# B&R Automation Studio project ai_powered_plc_development
Automation Studio 6.3.1.32; technology packages: mappConnect 6.1.0, mappView 6.1.1, OpcUaCs 6.0.0

## Configuration Main

CPU X20CP1686X, AutomationRuntime 6.3.3, Build 11.3.0, Vc 6.0.0

### Task classes (Cpu.sw)
```
Cyclic#1:
  method <- Method.method.prg
Cyclic#4:
  mco <- mco.prg
  Main <- Source.Main.prg
  Conveyor <- Source.Modules.Conveyor.Conveyor.prg
  Heater <- Source.Modules.Heater.Heater.prg
  Robot <- Source.Modules.Robot.Robot.prg
  AlarmHandl <- Source.Services.AlarmHandler.AlarmHandler.prg
Libraries: CoTrace, runtime, AsZip, FileIO, AsOpcUac, AsOpcUas
```

### Hardware
```
X20CP1686X : X20CP1686X v1.8.2.0
  Connector IF2:
    ActivateDevice = 1
  ConfigurationID = ai_powered_plc_development_mappConnectDemo
  AutomaticTransferOfUserfiles = on
  FileDevice1
  FileDeviceName1 = USER
  FileDevicePath1 = USER_PATH
  FileDevice2
  FileDeviceName2 = USER_web
  FileDevicePath2 = USER_PATH/web
  ActivateWebServer = 1
  WebServerProtocol = 1
```

### Config.mappconnect - X20CP1686X/mappConnect/Config.mappconnect
```
Element mapp Connect Configuration (Type=mappconnect)
  WebServerProtocol = 1
    WebServerPort = 8080
    Interface = All
    WebServerPortSsl = 8443
  WebServerEndpointConfiguration:
    Endpoint[1]  // Allow .html files for all users
      Endpoint = *.html
      Roles
    Endpoint[2]  // Allow stylesheet files for all users
      Endpoint = /css/*.css
      Roles
    Endpoint[3]  // Allow javascript files for all users
      Endpoint = /js/*.js
      Roles
    Endpoint[4]  // Allow all API endpoints for all users
      Endpoint = /api/1.0/*
      Roles
    Endpoint[5]  // Allow favicon and icon files
      Endpoint = *.ico
      Roles
    Endpoint[6]  // Allow common image types
      Endpoint = *.png
      Roles
    Endpoint[7]  // Allow common image types
      Endpoint = *.jpg
      Roles
    Endpoint[8]  // Allow common image types
      Endpoint = *.svg
      Roles
    Endpoint[9]  // Allow fonts
      Endpoint = *.woff2
      Roles
    Endpoint[10]  // Allow fonts
      Endpoint = *.woff
      Roles
    Endpoint[11]  // Allow fonts
      Endpoint = *.ttf
      Roles
    Endpoint[12]  // Allow source maps (dev)
      Endpoint = *.map
      Roles
    Endpoint[13]  // Allow typical asset folders
      Endpoint = /assets/*
      Roles
    Endpoint[14]  // Allow typical image folder
      Endpoint = /img/*
      Roles
    Endpoint[15]  // Allow additional static folder
      Endpoint = /static/*
      Roles
  OpcUaServerWhitelist:
    OpcUaServer[1]:
      Url = opc.tcp://127.0.0.1:4840
```

### AlarmCore.mpalarmxcore - X20CP1686X/mappServices/AlarmCore.mpalarmxcore
```
Element gAlarmXCore (Type=mpalarmxcore)
  mapp.Gen:
    Enable = TRUE
    EnableCockpit = TRUE
    TaskClass = 4
    Parent
  mapp.AlarmX.List:
    [0]:
      List = gAlarmXList
      Offset = 0
  mapp.AlarmX.Create = Disabled
  mapp.AlarmX.Core.Retain:
    Memory = 0
  mapp.AlarmX.Core.Categories:
    [0]:
      List = gAlarmXCategory
```

### AlarmHist.mpalarmxhistory - X20CP1686X/mappServices/AlarmHist.mpalarmxhistory
```
Element gAlarmXHistory (Type=mpalarmxhistory)
  mapp.Gen:
    Enable = TRUE
    EnableCockpit = TRUE
    Audit = TRUE
    Parent
  mapp.AlarmX.History:
    Export:
      TimeStampPattern = %Y-%m-%d %H:%M:%S:%L
      AutoExtension = TRUE
      ColumnSeparator = ,
    Memory = 0
      Size = 200
      BufferSize = 10
      Interval = 60
    Scope = 0
```

### AlarmList.mpalarmxlist - X20CP1686X/mappServices/AlarmList.mpalarmxlist
```
Element gAlarmXList (Type=mpalarmxlist)
  mapp.AlarmX.Snippets:
    AutoDetect = 1
      Language
```

## Logical view

Binary libraries used (declarations not repeated): operator, runtime, AsIecCon, astime, CoTrace, AsZip, FileIO, AsOpcUac, AsOpcUas


### Program Logical/mco (ANSIC)

#### Variables.var
```iecst
VAR
	myVar : LREAL := 12.3;
	myVar2 : REAL := 11;
END_VAR
```

#### compile_flags.txt
```
# This file is auto-generated by ASX. Do not edit manually, as changes may be overwritten.
# If you need to manually edit this file and prevent automatic updates, add "# MANUAL EDIT" to the first line.
-I
c:\projects\Private\ai_powered_plc_development\Logical\mco
-I
c:\projects\Private\ai_powered_plc_development\Temp\Includes\mco
-I
C:\Program Files (x86)\BRAutomation\AS6\AS\gnuinst\V11.3.0\6.0\i686-elf\include\c++\11.3.0
-I
C:\Program Files (x86)\BRAutomation\AS6\AS\gnuinst\V11.3.0\6.0\i686-elf\include\c++\11.3.0\i686-elf
-I
C:\Program Files (x86)\BRAutomation\AS6\AS\gnuinst\V11.3.0\6.0\i686-elf\include\c++\11.3.0\backward
-I
C:\Program Files (x86)\BRAutomation\AS6\AS\gnuinst\V11.3.0\6.0\lib\gcc\i686-elf\11.3.0\include
-I
C:\Program Files (x86)\BRAutomation\AS6\AS\gnuinst\V11.3.0\6.0\lib\gcc\i686-elf\11.3.0\include-fixed
-I
C:\Program Files (x86)\BRAutomation\AS6\AS\gnuinst\V11.3.0\6.0\i686-elf\include
-I
c:\projects\Private\ai_powered_plc_development\Temp\Includes
-trigraphs
-fno-asm
-D
_DEFAULT_INCLUDES
-D
_SG4
--target=i686-elf
-fPIC
-Wall
```

#### Cyclic.c
```c
#include <bur/plctypes.h>

#ifdef _DEFAULT_INCLUDES
	#include <AsDefault.h>
#endif

void _CYCLIC ProgramCyclic(void)
{

}
```

### Program Logical/Method/method (ANSIC)

#### Cyclic.c - Cyclic code
```c
#include <bur/plctypes.h>

#ifdef _DEFAULT_INCLUDES
	#include <AsDefault.h>
#endif

#include <string.h>

void _CYCLIC ProgramCyclic(void)
{
	switch(state)
	{
		case WaitForCall:
			UaSrv_MethodOperate_0.Action = UaMoa_CheckIsCalled;
			UaSrv_MethodOperate(&UaSrv_MethodOperate_0);
			UaSrv_MethodOperate_0.Execute = !UaSrv_MethodOperate_0.Busy;
			if (UaSrv_MethodOperate_0.Done && UaSrv_MethodOperate_0.IsCalled)
			{
				state = ExecuteMethod;
			}
			if (UaSrv_MethodOperate_0.Error)
			{
				state = Error;
			}
			break;

		case ExecuteMethod:
			methodCalled = 1;
			output1 = input1 + input2;
			state = FinishMethod;
			UaSrv_MethodOperate_0.Execute = 1;
			break;

		case FinishMethod:
			UaSrv_MethodOperate_0.Action = UaMoa_Finished;
			UaSrv_MethodOperate(&UaSrv_MethodOperate_0);
			UaSrv_MethodOperate_0.Execute = !UaSrv_MethodOperate_0.Busy;
			if (UaSrv_MethodOperate_0.Done)
			{
				state = WaitForCall;
			}
			if (UaSrv_MethodOperate_0.Error)
			{
				state = Error;
			}
			break;

		case Error:
			break;

		default:
			state = Error;
	}
}
```

#### Types.typ - Local data types
```iecst
TYPE
	State :
		(
		WaitForCall,
		ExecuteMethod,
		FinishMethod,
		Error
		);
END_TYPE
```

#### Variables.var - Local variables
```iecst
VAR
	output1 : DINT;
	input1 : DINT;
	UaSrv_MethodOperate_0 : UaSrv_MethodOperate;
	state : State := WaitForCall;
END_VAR
VAR CONSTANT
	cMethodName : STRING[32] := 'add';
END_VAR
VAR
	methodCalled : BOOL := FALSE;
	input2 : DINT;
END_VAR
```

- Methods.uam (not shown)

#### Init.c - Initialization code
```c
#include <bur/plctypes.h>

#ifdef _DEFAULT_INCLUDES
	#include <AsDefault.h>
#endif

#include <string.h>

void _INIT ProgramInit(void)
{
	strcpy(UaSrv_MethodOperate_0.MethodName, cMethodName);
}
```

### MainIface.typ
```iecst
TYPE
	MainCmdIfaceType : STRUCT
		Start : BOOL;
		Stop  : BOOL;
	END_STRUCT;

	MainParIfaceType : STRUCT
		Reserved : BOOL;
	END_STRUCT;

	MainStatusIfaceType : STRUCT
		State       : STRING[32];
		Substate    : STRING[32];
		LineRunning : BOOL;
		AnyFault    : BOOL;
	END_STRUCT;

	MainIfaceType : STRUCT
		Cmd    : MainCmdIfaceType;
		Par    : MainParIfaceType;
		Status : MainStatusIfaceType;
	END_STRUCT;
END_TYPE
```

### MainIface.var
```iecst
VAR
	gMain : MainIfaceType;
END_VAR

VAR CONSTANT

END_VAR
```

### Types.typ
```iecst
TYPE
	(* HMI data transfer objects for Main aggregate *)

	ConveyorHmiData : STRUCT
		Running    : BOOL;
		Fault      : BOOL;
		Speed      : REAL;      (* m/s *)
		Load       : REAL;      (* % *)
		PartsCount : UDINT;
		Mode       : STRING[16];
	END_STRUCT;

	HeaterHmiData : STRUCT
		Heating      : BOOL;
		Fault        : BOOL;
		Temperature  : REAL;     (* °C *)
		PowerPercent : REAL;     (* % *)
		Setpoint     : REAL;     (* °C *)
	END_STRUCT;

	RobotHmiData : STRUCT
		Auto  : BOOL;
		Fault : BOOL;
		X     : REAL;
		Y     : REAL;
		Z     : REAL;
		State : STRING[32];
	END_STRUCT;

	MachineCommandsType : STRUCT
		Start : BOOL;
		Stop  : BOOL;
	END_STRUCT;

	MachineHmiData : STRUCT
		State       : STRING[32];
		Substate    : STRING[64];
		LineRunning : BOOL;
		AnyFault    : BOOL;
		Conveyor    : ConveyorHmiData;
		Heater      : HeaterHmiData;
		Robot       : RobotHmiData;
		Commands    : MachineCommandsType;
	END_STRUCT;

END_TYPE
```

### Variables.var
```iecst
VAR
    MachineHmi : MachineHmiData; (* Exposed HMI aggregate *)
    runRequest : BOOL; (* internal latched run flag *)
END_VAR

VAR CONSTANT

END_VAR
```

### MainIface.typ - not listed in the package file held
```iecst
TYPE
    MainCmdIfaceType : STRUCT
        Start : BOOL;
        Stop  : BOOL;
    END_STRUCT;

    MainParIfaceType : STRUCT
        Reserved : BOOL;
    END_STRUCT;

    MainStatusIfaceType : STRUCT
        State     : STRING[32];
        Substate  : STRING[32];
        LineRunning : BOOL;
        AnyFault    : BOOL;
    END_STRUCT;

    MainIfaceType : STRUCT
        Cmd    : MainCmdIfaceType;
        Par    : MainParIfaceType;
        Status : MainStatusIfaceType;
    END_STRUCT;
END_TYPE
```

### MainIface.var - not listed in the package file held
```iecst
VAR
    gMain : MainIfaceType;
END_VAR

VAR CONSTANT
END_VAR
```

### Main.st - not listed in the package file held
```iecst
PROGRAM _INIT
	(* Insert code here *)
	(* Initialize defaults *)
	MachineHmi.LineRunning := FALSE;
	MachineHmi.State := 'Idle';
	MachineHmi.Substate := '';
	runRequest := FALSE;
	(* Initialize main interface status *)
	gMain.Status.State := 'Idle';
	gMain.Status.Substate := '';
	gMain.Status.LineRunning := FALSE;
	gMain.Status.AnyFault := FALSE;
END_PROGRAM

PROGRAM _CYCLIC
	(* Pull conveyor status from its program interface *)
	MachineHmi.Conveyor.Running := gConveyor.Status.Running;
	MachineHmi.Conveyor.Fault := gConveyor.Status.Fault;
	MachineHmi.Conveyor.Speed := gConveyor.Status.Speed_mps;
	MachineHmi.Conveyor.Load := gConveyor.Status.Load_pct;
	MachineHmi.Conveyor.PartsCount := gConveyor.Status.PartsCount;
	MachineHmi.Conveyor.Mode := gConveyor.Status.Mode;

	(* Heater status from module interface *)
	MachineHmi.Heater.Heating := gHeater.Status.Heating;
	MachineHmi.Heater.Fault := gHeater.Status.Fault;
	MachineHmi.Heater.Temperature := gHeater.Status.TemperatureC;
	MachineHmi.Heater.PowerPercent := gHeater.Status.Power_pct;
	IF gHeater.Par.Setpoint_C <> 0.0 THEN MachineHmi.Heater.Setpoint := gHeater.Par.Setpoint_C; END_IF;

	(* Robot status from module interface *)
	MachineHmi.Robot.Auto := gRobot.Status.Auto;
	MachineHmi.Robot.Fault := gRobot.Status.Fault;
	MachineHmi.Robot.X := gRobot.Status.X;
	MachineHmi.Robot.Y := gRobot.Status.Y;
	MachineHmi.Robot.Z := gRobot.Status.Z;
	MachineHmi.Robot.State := gRobot.Status.State;

	(* Aggregate HMI level flags *)
	MachineHmi.AnyFault := MachineHmi.Conveyor.Fault OR MachineHmi.Heater.Fault OR MachineHmi.Robot.Fault;
	MachineHmi.LineRunning := runRequest AND NOT MachineHmi.AnyFault;

	(* Interfaces already mapped above *)

	(* Determine State/Substate *)
	IF MachineHmi.AnyFault THEN
		MachineHmi.State := 'Fault';
		MachineHmi.Substate := 'Check modules';
	ELSIF runRequest THEN
		MachineHmi.State := 'Auto';
		IF NOT gConveyor.Status.Running THEN
			MachineHmi.Substate := 'Starting conveyor';
		ELSIF NOT gRobot.Status.Auto THEN
			MachineHmi.Substate := 'Starting robot';
		ELSE
			MachineHmi.Substate := 'Production';
		END_IF;
	ELSE
		MachineHmi.State := 'Idle';
		MachineHmi.Substate := 'Waiting for start';
	END_IF;

	(* Process Commands from HMI *)
	IF MachineHmi.Commands.Start THEN
		runRequest := TRUE;
	END_IF;
	IF MachineHmi.Commands.Stop THEN
		runRequest := FALSE;
	END_IF;
	(* auto-clear command bits to behave as pulses *)
	MachineHmi.Commands.Start := FALSE;
	MachineHmi.Commands.Stop := FALSE;

	(* Update global main interface *)
	gMain.Status.State := MachineHmi.State;
	gMain.Status.Substate := MachineHmi.Substate;
	gMain.Status.LineRunning := MachineHmi.LineRunning;
	gMain.Status.AnyFault := MachineHmi.AnyFault;

	(* Accept commands via gMain as well *)
	IF gMain.Cmd.Start THEN runRequest := TRUE; END_IF;
	IF gMain.Cmd.Stop THEN runRequest := FALSE; END_IF;
	gMain.Cmd.Start := FALSE;
	gMain.Cmd.Stop := FALSE;
END_PROGRAM

PROGRAM _EXIT
	(* Insert code here *)

END_PROGRAM
```

### Program Logical/Source/Modules/Heater (IEC)

#### Heater.st - Init, cyclic, exit code
```iecst
(* Moved to Modules/Heater/Heater/Heater.st — not used. Keep for reference only. *)
PROGRAM _INIT
	IF gHeater.Par.Setpoint_C = 0.0 THEN gHeater.Par.Setpoint_C := 180.0; END_IF;
END_PROGRAM

PROGRAM _CYCLIC
	(* Oscillate temperature around setpoint and compute power *)
	IF heaterUp THEN
		gHeater.Status.TemperatureC := gHeater.Status.TemperatureC + 0.5;
		IF gHeater.Status.TemperatureC >= gHeater.Par.Setpoint_C + 5.0 THEN heaterUp := FALSE; END_IF;
	ELSE
		gHeater.Status.TemperatureC := gHeater.Status.TemperatureC - 0.5;
		IF gHeater.Status.TemperatureC <= gHeater.Par.Setpoint_C - 5.0 THEN heaterUp := TRUE; END_IF;
	END_IF;
	gHeater.Status.Heating := gHeater.Status.TemperatureC < gHeater.Par.Setpoint_C;
	IF gHeater.Status.Heating THEN
		gHeater.Status.Power_pct := 60.0;
	ELSE
		gHeater.Status.Power_pct := 10.0;
	END_IF;
	gHeater.Status.Fault := FALSE;
END_PROGRAM

PROGRAM _EXIT
END_PROGRAM
```

#### Variables.var - Local variables
```iecst
VAR
    heaterUp : BOOL := TRUE;
END_VAR

VAR CONSTANT
END_VAR
```

#### HeaterIface.typ - not listed in the package file held
```iecst
TYPE
    HeaterCmdIfaceType : STRUCT
        Enable : BOOL;
    END_STRUCT;

    HeaterParIfaceType : STRUCT
        Setpoint_C : REAL := 180.0;
    END_STRUCT;

    HeaterStatusIfaceType : STRUCT
        Heating      : BOOL;
        Fault        : BOOL;
        TemperatureC : REAL;
        Power_pct    : REAL;
    END_STRUCT;

    HeaterIfaceType : STRUCT
        Cmd    : HeaterCmdIfaceType;
        Par    : HeaterParIfaceType;
        Status : HeaterStatusIfaceType;
    END_STRUCT;
END_TYPE
```

#### Program Logical/Source/Modules/Heater/Heater

##### Heater.st
```iecst
PROGRAM _INIT
	IF gHeater.Par.Setpoint_C = 0.0 THEN gHeater.Par.Setpoint_C := 180.0; END_IF;
END_PROGRAM

PROGRAM _CYCLIC
	(* Oscillate temperature around setpoint and compute power *)
	IF heaterUp THEN
		gHeater.Status.TemperatureC := gHeater.Status.TemperatureC + 0.5;
		IF gHeater.Status.TemperatureC >= gHeater.Par.Setpoint_C + 5.0 THEN heaterUp := FALSE; END_IF;
	ELSE
		gHeater.Status.TemperatureC := gHeater.Status.TemperatureC - 0.5;
		IF gHeater.Status.TemperatureC <= gHeater.Par.Setpoint_C - 5.0 THEN heaterUp := TRUE; END_IF;
	END_IF;
	gHeater.Status.Heating := gHeater.Status.TemperatureC < gHeater.Par.Setpoint_C;
	IF gHeater.Status.Heating THEN
		gHeater.Status.Power_pct := 60.0;
	ELSE
		gHeater.Status.Power_pct := 10.0;
	END_IF;
	gHeater.Status.Fault := FALSE;
END_PROGRAM

PROGRAM _EXIT
END_PROGRAM
```

### Program Logical/Source/Modules/Robot (IEC)

#### Robot.st - Init, cyclic, exit code
```iecst
(* Moved to Modules/Robot/Robot/Robot.st — not used. Keep for reference only. *)

PROGRAM _INIT
	(* Initialize to a known state *)
	gRobot.Status.State := 'Homing';
	gRobot.Status.Auto := FALSE;
	gRobot.Status.X := 0.0; gRobot.Status.Y := 0.0; gRobot.Status.Z := 0.0;
	robotStep := 1;
END_PROGRAM

PROGRAM _CYCLIC
	(* Simple motion pattern and state machine *)
	CASE robotStep OF
		1: gRobot.Status.State := 'Auto'; gRobot.Status.Auto := TRUE; gRobot.Status.X := gRobot.Status.X + 1.0; IF gRobot.Status.X >= 100.0 THEN robotStep := 2; END_IF;
		2: gRobot.Status.Y := gRobot.Status.Y + 1.0; IF gRobot.Status.Y >= 50.0 THEN robotStep := 3; END_IF;
		3: gRobot.Status.X := gRobot.Status.X - 1.0; IF gRobot.Status.X <= 0.0 THEN robotStep := 4; END_IF;
		4: gRobot.Status.Y := gRobot.Status.Y - 1.0; IF gRobot.Status.Y <= 0.0 THEN robotStep := 1; END_IF;
	END_CASE;
	gRobot.Status.Fault := FALSE;
END_PROGRAM

PROGRAM _EXIT
END_PROGRAM
```

#### Variables.var - Local variables
```iecst
VAR
    robotStep : INT;
END_VAR

VAR CONSTANT
END_VAR
```

#### RobotIface.var - not listed in the package file held
```iecst
VAR
    gRobot : RobotIfaceType;
END_VAR

VAR CONSTANT
END_VAR
```

#### Program Logical/Source/Modules/Robot/Robot

##### Robot.st
```iecst
PROGRAM _INIT
	(* Initialize to a known state *)
	gRobot.Status.State := 'Homing';
	gRobot.Status.Auto := FALSE;
	gRobot.Status.X := 0.0; gRobot.Status.Y := 0.0; gRobot.Status.Z := 0.0;
	robotStep := 1;
END_PROGRAM

PROGRAM _CYCLIC
	(* Simple motion pattern and state machine *)
	CASE robotStep OF
		1: gRobot.Status.State := 'Auto'; gRobot.Status.Auto := TRUE; gRobot.Status.X := gRobot.Status.X + 1.0; IF gRobot.Status.X >= 100.0 THEN robotStep := 2; END_IF;
		2: gRobot.Status.Y := gRobot.Status.Y + 1.0; IF gRobot.Status.Y >= 50.0 THEN robotStep := 3; END_IF;
		3: gRobot.Status.X := gRobot.Status.X - 1.0; IF gRobot.Status.X <= 0.0 THEN robotStep := 4; END_IF;
		4: gRobot.Status.Y := gRobot.Status.Y - 1.0; IF gRobot.Status.Y <= 0.0 THEN robotStep := 1; END_IF;
	END_CASE;
	gRobot.Status.Fault := FALSE;
END_PROGRAM

PROGRAM _EXIT
END_PROGRAM
```

### Program Logical/Source/Modules/Conveyor (IEC)

#### ConveyorIface.var - not listed in the package file held
```iecst
VAR
    gConveyor : ConveyorIfaceType;
END_VAR

VAR CONSTANT
END_VAR
```

#### Program Logical/Source/Modules/Conveyor/Conveyor (IEC)

##### Conveyor.st - Init, cyclic, exit code
```iecst
PROGRAM _INIT
	(* Initialize interface defaults if needed *)
	gConveyor.Status.Mode := 'AUTO';
END_PROGRAM

PROGRAM _CYCLIC
	(* Simple simulation: ramp speed 0..2 m/s and load 0..100%, toggle dir, increment parts *)
	IF convUp THEN
		gConveyor.Status.Speed_mps := gConveyor.Status.Speed_mps + 0.02;
		gConveyor.Status.Load_pct := gConveyor.Status.Load_pct + 1.0;
		IF gConveyor.Status.Speed_mps >= 2.0 THEN convUp := FALSE; END_IF;
	ELSE
		gConveyor.Status.Speed_mps := gConveyor.Status.Speed_mps - 0.02;
		gConveyor.Status.Load_pct := gConveyor.Status.Load_pct - 1.0;
		IF gConveyor.Status.Speed_mps <= 0.0 THEN convUp := TRUE; END_IF;
	END_IF;

	IF gConveyor.Status.Load_pct < 0.0 THEN gConveyor.Status.Load_pct := 0.0; END_IF;
	IF gConveyor.Status.Load_pct > 100.0 THEN gConveyor.Status.Load_pct := 100.0; END_IF;

	gConveyor.Status.Running := TRUE;
	convCnt := convCnt + 1;
	IF (convCnt MOD 50) = 0 THEN
		gConveyor.Status.PartsCount := gConveyor.Status.PartsCount + 1;
	END_IF;
	gConveyor.Status.Fault := FALSE;
END_PROGRAM

PROGRAM _EXIT
END_PROGRAM
```

##### Variables.var - Local variables
```iecst
VAR
    convCnt : UDINT;
    convUp  : BOOL := TRUE;
END_VAR

VAR CONSTANT
END_VAR
```

### ConveyorIface.typ - not listed in the package file held
```iecst
TYPE
    ConveyorCmdIfaceType : STRUCT
        Start : BOOL;
        Stop  : BOOL;
    END_STRUCT;

    ConveyorParIfaceType : STRUCT
        MaxSpeed_mps : REAL := 2.0;
    END_STRUCT;

    ConveyorStatusIfaceType : STRUCT
        Running    : BOOL;
        Fault      : BOOL;
        Speed_mps  : REAL;
        Load_pct   : REAL;
        PartsCount : DINT;
        Mode       : STRING[32];
    END_STRUCT;

    ConveyorIfaceType : STRUCT
        Cmd    : ConveyorCmdIfaceType;
        Par    : ConveyorParIfaceType;
        Status : ConveyorStatusIfaceType;
    END_STRUCT;
END_TYPE
```

### RobotIface.typ - not listed in the package file held
```iecst
TYPE
    RobotCmdIfaceType : STRUCT
        Auto : BOOL;
    END_STRUCT;

    RobotParIfaceType : STRUCT
        Speed_pct : REAL := 50.0;
    END_STRUCT;

    RobotStatusIfaceType : STRUCT
        Auto   : BOOL;
        Fault  : BOOL;
        X      : REAL;
        Y      : REAL;
        Z      : REAL;
        State  : STRING[32];
    END_STRUCT;

    RobotIfaceType : STRUCT
        Cmd    : RobotCmdIfaceType;
        Par    : RobotParIfaceType;
        Status : RobotStatusIfaceType;
    END_STRUCT;
END_TYPE
```

### Types.typ - not listed in the package file held
```iecst
TYPE
	ConveyorHmiData : STRUCT
		Running : BOOL;
		Fault : BOOL;
		Speed : REAL; (* m/s *)
		Load : REAL;  (* % *)
		PartsCount : DINT;
		Mode : STRING[32];
	END_STRUCT;

	HeaterHmiData : STRUCT
		Heating : BOOL;
		Fault : BOOL;
		Temperature : REAL; (* °C *)
		Setpoint : REAL;    (* °C *)
		PowerPercent : REAL; (* % *)
	END_STRUCT;

	RobotHmiData : STRUCT
		Auto : BOOL;
		Fault : BOOL;
		X : REAL;
		Y : REAL;
		Z : REAL;
		State : STRING[32];
	END_STRUCT;

	MachineHmiData : STRUCT
		Conveyor : ConveyorHmiData;
		Heater : HeaterHmiData;
		Robot : RobotHmiData;
		LineRunning : BOOL;
		AnyFault : BOOL;
		State : STRING[32];
		Substate : STRING[32];
		Commands : STRUCT
			Start : BOOL;
			Stop : BOOL;
		END_STRUCT;
	END_STRUCT;
END_TYPE
```

### HeaterIface.var - not listed in the package file held
```iecst
VAR
    gHeater : HeaterIfaceType;
END_VAR

VAR CONSTANT
END_VAR
```

### Conveyor.st - not listed in the package file held
```iecst
PROGRAM _INIT
	(* Initialization for Conveyor module *)
END_PROGRAM

PROGRAM _CYCLIC
	(* Not used for module; logic in Function Block *)
END_PROGRAM

FUNCTION_BLOCK FB_Conveyor
	VAR
		Hmi : ConveyorHmiData; (* Variables to expose on HMI *)
		cnt : UDINT;
		up : BOOL := TRUE;
	END_VAR

	(* Simple simulation: ramp speed 0..2 m/s and load 0..100%, toggle running, increment parts *)
	IF up THEN
		Hmi.Speed := Hmi.Speed + 0.02;
		Hmi.Load := Hmi.Load + 1.0;
		IF Hmi.Speed >= 2.0 THEN up := FALSE; END_IF;
	ELSE
		Hmi.Speed := Hmi.Speed - 0.02;
		Hmi.Load := Hmi.Load - 1.0;
		IF Hmi.Speed <= 0.0 THEN up := TRUE; END_IF;
	END_IF;
	IF Hmi.Load < 0.0 THEN Hmi.Load := 0.0; END_IF;
	IF Hmi.Load > 100.0 THEN Hmi.Load := 100.0; END_IF;

	Hmi.Running := TRUE;
	Hmi.Mode := 'AUTO';
	cnt := cnt + 1;
	IF (cnt MOD 50) = 0 THEN
		Hmi.PartsCount := Hmi.PartsCount + 1;
	END_IF;
	Hmi.Fault := FALSE;
	(* Reflect into global interface *)
	gConveyor.Status.Running := Hmi.Running;
	gConveyor.Status.Fault := Hmi.Fault;
	gConveyor.Status.Speed_mps := Hmi.Speed;
	gConveyor.Status.Load_pct := Hmi.Load;
	gConveyor.Status.PartsCount := Hmi.PartsCount;
	gConveyor.Status.Mode := Hmi.Mode;
END_FUNCTION_BLOCK
```

### Heater.st - not listed in the package file held
```iecst
PROGRAM _INIT
	(* Initialization for Heater module *)
END_PROGRAM

PROGRAM _CYCLIC
	(* Not used for module; logic in Function Block *)
END_PROGRAM

FUNCTION_BLOCK FB_Heater
	VAR
		Hmi : HeaterHmiData; (* Variables to expose on HMI *)
		up : BOOL := TRUE;
	END_VAR

	(* Simple simulation: oscillate temperature around setpoint and power percent *)
	IF Hmi.Setpoint = 0.0 THEN Hmi.Setpoint := 180.0; END_IF;
	IF up THEN
		Hmi.Temperature := Hmi.Temperature + 0.5;
		IF Hmi.Temperature >= Hmi.Setpoint + 5.0 THEN up := FALSE; END_IF;
	ELSE
		Hmi.Temperature := Hmi.Temperature - 0.5;
		IF Hmi.Temperature <= Hmi.Setpoint - 5.0 THEN up := TRUE; END_IF;
	END_IF;
	Hmi.Heating := Hmi.Temperature < Hmi.Setpoint;
	IF Hmi.Heating THEN
		Hmi.PowerPercent := 60.0;
	ELSE
		Hmi.PowerPercent := 10.0;
	END_IF;
	Hmi.Fault := FALSE;
	(* Reflect into global interface *)
	gHeater.Status.Heating := Hmi.Heating;
	gHeater.Status.Fault := Hmi.Fault;
	gHeater.Status.TemperatureC := Hmi.Temperature;
	gHeater.Status.Power_pct := Hmi.PowerPercent;
	IF Hmi.Setpoint <> 0.0 THEN gHeater.Par.Setpoint_C := Hmi.Setpoint; END_IF;
END_FUNCTION_BLOCK
```

### Robot.st - not listed in the package file held
```iecst
PROGRAM _INIT
	(* Initialization for Robot module *)
END_PROGRAM

PROGRAM _CYCLIC
	(* Not used for module; logic in Function Block *)
END_PROGRAM

FUNCTION_BLOCK FB_Robot
	VAR
		Hmi : RobotHmiData; (* Variables to expose on HMI *)
		step : INT;
	END_VAR

	(* Simple simulation: move in a square path and cycle through states *)
	CASE step OF
		0: Hmi.State := 'Homing'; Hmi.Auto := FALSE; Hmi.X := 0.0; Hmi.Y := 0.0; Hmi.Z := 0.0; step := 1;
		1: Hmi.State := 'Auto'; Hmi.Auto := TRUE; Hmi.X := Hmi.X + 1.0; IF Hmi.X >= 100.0 THEN step := 2; END_IF;
		2: Hmi.Y := Hmi.Y + 1.0; IF Hmi.Y >= 50.0 THEN step := 3; END_IF;
		3: Hmi.X := Hmi.X - 1.0; IF Hmi.X <= 0.0 THEN step := 4; END_IF;
		4: Hmi.Y := Hmi.Y - 1.0; IF Hmi.Y <= 0.0 THEN step := 1; END_IF;
	END_CASE;
	Hmi.Fault := FALSE;
	(* Reflect into global interface *)
	gRobot.Status.Auto := Hmi.Auto;
	gRobot.Status.Fault := Hmi.Fault;
	gRobot.Status.X := Hmi.X;
	gRobot.Status.Y := Hmi.Y;
	gRobot.Status.Z := Hmi.Z;
	gRobot.Status.State := Hmi.State;
END_FUNCTION_BLOCK
```

### AlarmHandlerIface.typ
```iecst
TYPE
    AlarmHandlerCmdIfaceType : STRUCT
        AckAll          : BOOL;
        ResetAll        : BOOL;
        SilenceHorn     : BOOL;
        ShelveSelected  : BOOL;
        UnshelveAll     : BOOL;
        SelectFirstUnacked : BOOL;
    END_STRUCT;

    AlarmHandlerParIfaceType : STRUCT
        EnableHistory   : BOOL := TRUE;
        MaxLocalLog     : UINT := 64;
    END_STRUCT;

    AlarmRecordType : STRUCT
        Code       : DINT;
        Severity   : USINT;
        Active     : BOOL;
        Acknowledged : BOOL;
        Timestamp  : UDINT;
    END_STRUCT;

    AlarmHandlerStatusIfaceType : STRUCT
        ActiveCount      : UINT;
        UnackedCount     : UINT;
        HighestSeverity  : USINT;
        AnyActive        : BOOL;
        AnyUnacked       : BOOL;
        Log              : ARRAY[0..63] OF AlarmRecordType;
        LogSize          : UINT;
    END_STRUCT;

    AlarmHandlerIfaceType : STRUCT
        Cmd    : AlarmHandlerCmdIfaceType;
        Par    : AlarmHandlerParIfaceType;
        Status : AlarmHandlerStatusIfaceType;
    END_STRUCT;
END_TYPE
```

### AlarmHandlerIface.var
```iecst
VAR
	gAlarmHandler : AlarmHandlerIfaceType;
END_VAR

VAR CONSTANT
	(* Reserved for severities/codes mapping if needed later *)
END_VAR
```

### Program Logical/Source/Services/AlarmHandler/AlarmHandler (IEC)

#### Variables.var
```iecst
VAR
	logHead : UINT;        (* ring buffer head index [0..63] *)
	demoTick : UDINT;      (* demo timer for possible test alarms *)
END_VAR
```

#### Main.st
```iecst
PROGRAM _INIT
	// Initialize counters
	gAlarmHandler.Status.ActiveCount := 0;
	gAlarmHandler.Status.UnackedCount := 0;
	gAlarmHandler.Status.HighestSeverity := 0;
	gAlarmHandler.Status.AnyActive := FALSE;
	gAlarmHandler.Status.AnyUnacked := FALSE;
	gAlarmHandler.Status.LogSize := 0;
END_PROGRAM

PROGRAM _CYCLIC
	// Demo-only core
	// In a real build, you would call mapp AlarmX FBs (MpAlarmXCore, MpAlarmXHistory) here.
	// We keep a small local ring buffer for HMI quick summaries.

	// Handle commands (edge tolerant simple reset)
	IF gAlarmHandler.Cmd.AckAll THEN
		// TODO: MpAlarmXAckAll() via appropriate FB call
		gAlarmHandler.Cmd.AckAll := FALSE;
	END_IF;
	IF gAlarmHandler.Cmd.ResetAll THEN
		// TODO: MpAlarmXResetAll()
		gAlarmHandler.Cmd.ResetAll := FALSE;
	END_IF;
	IF gAlarmHandler.Cmd.SilenceHorn THEN
		gAlarmHandler.Cmd.SilenceHorn := FALSE;
	END_IF;
	IF gAlarmHandler.Cmd.ShelveSelected THEN
		gAlarmHandler.Cmd.ShelveSelected := FALSE;
	END_IF;
	IF gAlarmHandler.Cmd.UnshelveAll THEN
		gAlarmHandler.Cmd.UnshelveAll := FALSE;
	END_IF;

	// Example: simulate a trivial status rollup (replace with MpAlarmXCore statistics)
	// Keep values as-is; HMI can still bind. Real counts come from mapp in production.

	// Optional: local log maintenance bounded by Par.MaxLocalLog
	IF gAlarmHandler.Par.EnableHistory THEN
		IF gAlarmHandler.Status.LogSize > gAlarmHandler.Par.MaxLocalLog THEN
			gAlarmHandler.Status.LogSize := gAlarmHandler.Par.MaxLocalLog;
		END_IF;
	END_IF;
END_PROGRAM

PROGRAM _EXIT
END_PROGRAM
```

### AlarmHanderIface.typ - not listed in the package file held
```iecst
TYPE
	AlarmHandlerCmdIfaceType : STRUCT
		AckAll          : BOOL;  (* Acknowledge all acknowledgeable alarms *)
		ResetAll        : BOOL;  (* Reset all resettable alarms *)
		SilenceHorn     : BOOL;  (* Example: mute buzzer *)
		ShelveSelected  : BOOL;  (* Shelve current selection (if supported) *)
		UnshelveAll     : BOOL;
		SelectFirstUnacked : BOOL; (* UI helper: request selection of first unacked *)
	END_STRUCT;

	AlarmHandlerParIfaceType : STRUCT
		EnableHistory   : BOOL := TRUE;  (* if TRUE, collect a ring buffer locally *)
		MaxLocalLog     : UINT := 64;    (* local circular buffer size *)
	END_STRUCT;

	AlarmRecordType : STRUCT
		Code       : DINT;
		Severity   : USINT;   (* 0..255 mapping to Info..Critical *)
		Active     : BOOL;
		Acknowledged : BOOL;
		Timestamp  : UDINT;   (* ms since boot; for demo *)
	END_STRUCT;

	AlarmHandlerStatusIfaceType : STRUCT
		ActiveCount      : UINT;
		UnackedCount     : UINT;
		HighestSeverity  : USINT;
		AnyActive        : BOOL;
		AnyUnacked       : BOOL;
		(* Local buffer for HMI quick view *)
		Log              : ARRAY[0..63] OF AlarmRecordType; (* truncated by MaxLocalLog *)
		LogSize          : UINT;
	END_STRUCT;

	AlarmHandlerIfaceType : STRUCT
		Cmd    : AlarmHandlerCmdIfaceType;
		Par    : AlarmHandlerParIfaceType;
		Status : AlarmHandlerStatusIfaceType;
	END_STRUCT;
END_TYPE
```

Listed in the project but not available here: Logical/Global.typ, Logical/Global.var, Logical/Method/method/Exit.c, Logical/Source/Main/Main, Logical/Source/Modules/Heater/Types.typ, Logical/Source/Modules/Conveyor/Conveyor.st, Logical/Source/Modules/Conveyor/Variables.var, Logical/Source/Modules/Conveyor/Conveyor/Types.typ, Logical/Package1
